# EPICS IOC start-up script: iocsh/iocStats.iocsh
dbLoadRecords("iocAdminSoft-ess.db", "IOC=$(IOCNAME)")
